// SIMATIC S7-200 SMART project (STEP 7-Micro/WIN SMART), CPU ST40

SYMBOL_TABLE Table 1
Counter_1        C1
UDP_Done         M0.0
UDP_Busy         M0.1
UDP_Error        M0.2
UDP_Stat         MB1
SEND_Done        M2.0
SEND_Busy        M2.1
SEND_Error       M2.2
SEND_Stat        MB3
REC_Done         M4.0
REC_Busy         M4.1
REC_Error        M4.2
REC_Stat         MB5
REC_Len          MW6
REC_IP1          MB8
REC_IP2          MB9
REC_IP3          MB10
REC_IP4          MB11
REC_RemPort      MW12
ConnID           MW14
LocPort          MW16
RemPort          MW18
END_SYMBOL_TABLE

SYMBOL_TABLE System Symbols
Always_On        SM0.0    // Always ON
First_Scan_On    SM0.1    // ON for the first scan cycle only
Clock_1s         SM0.5    // Clock pulse that is ON for 0.5 s, OFF for 0.5 s, for a duty cycle time of 1 s.
END_SYMBOL_TABLE

ORGANIZATION_BLOCK MAIN:OB1
TITLE=Program Comments
BEGIN
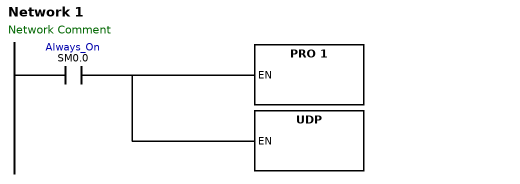
Network 1
// Network Comment
LD     Always_On:SM0.0
CALL   PRO 1:SBR0
CALL   UDP:SBR10
END_ORGANIZATION_BLOCK

SUBROUTINE_BLOCK PRO 1:SBR0
TITLE=
BEGIN
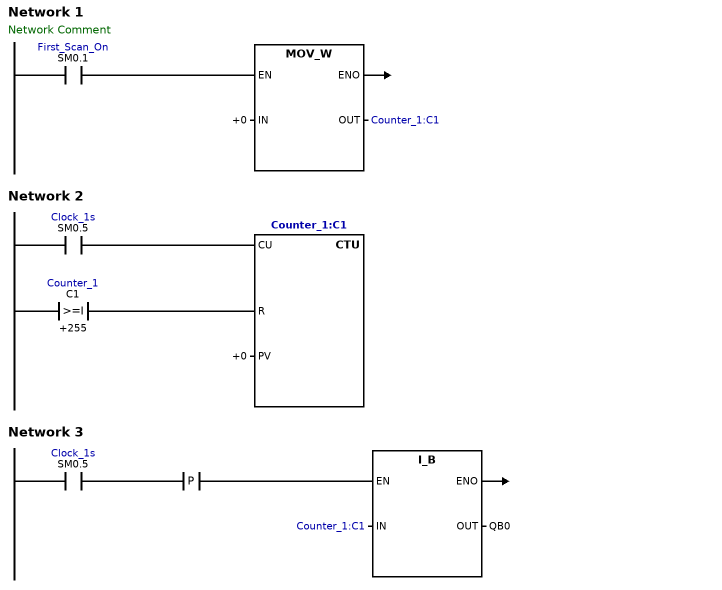
Network 1
// Network Comment
LD     First_Scan_On:SM0.1
MOVW   +0, Counter_1:C1
Network 2
LD     Clock_1s:SM0.5
LDW>=  Counter_1:C1, +255
CTU    Counter_1:C1, +0
Network 3
LD     Clock_1s:SM0.5
EU
ITB    Counter_1:C1, QB0
END_SUBROUTINE_BLOCK

SUBROUTINE_BLOCK UDP:SBR10
TITLE=Subroutine Comments
BEGIN
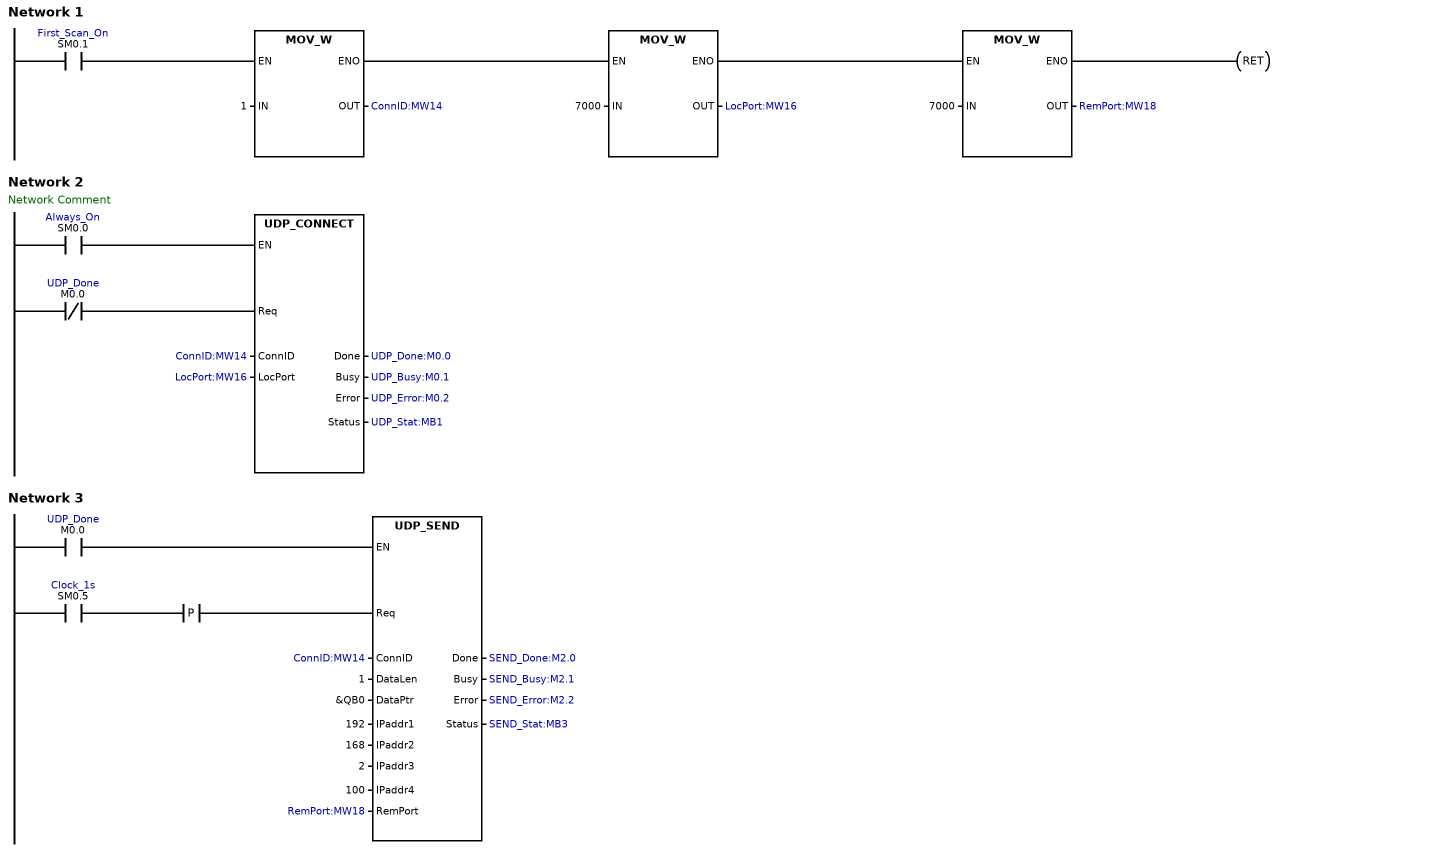
Network 1
LD     First_Scan_On:SM0.1
MOVW   1, ConnID:MW14
AENO
MOVW   7000, LocPort:MW16
AENO
MOVW   7000, RemPort:MW18
AENO
CRET
Network 2
// Network Comment
LD     Always_On:SM0.0
=      L60.0
LDN    UDP_Done:M0.0
=      L63.7
LD     L60.0
CALL   UDP_CONNECT:SBR11, L63.7, ConnID:MW14, LocPort:MW16, UDP_Done:M0.0, UDP_Busy:M0.1, UDP_Error:M0.2, UDP_Stat:MB1
Network 3
LD     UDP_Done:M0.0
=      L60.0
LD     Clock_1s:SM0.5
EU
=      L63.7
LD     L60.0
CALL   UDP_SEND:SBR12, L63.7, ConnID:MW14, 1, &QB0, 192, 168, 2, 100, RemPort:MW18, SEND_Done:M2.0, SEND_Busy:M2.1, SEND_Error:M2.2, SEND_Stat:MB3
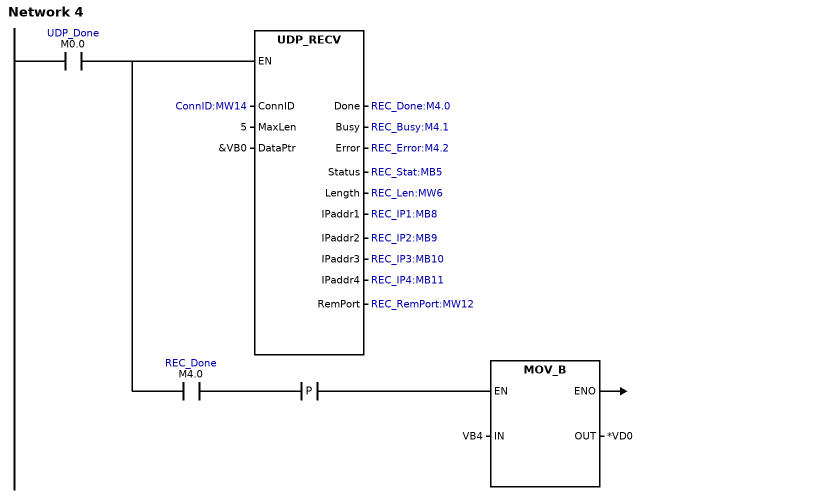
Network 4
LD     UDP_Done:M0.0
CALL   UDP_RECV:SBR13, ConnID:MW14, 5, &VB0, REC_Done:M4.0, REC_Busy:M4.1, REC_Error:M4.2, REC_Stat:MB5, REC_Len:MW6, REC_IP1:MB8, REC_IP2:MB9, REC_IP3:MB10, REC_IP4:MB11, REC_RemPort:MW12
A      REC_Done:M4.0
EU
MOVB   VB4, *VD0
END_SUBROUTINE_BLOCK

// SBR11: protected block, not included

// SBR12: protected block, not included

// SBR13: protected block, not included
